{attribute 'GeneratedUsingTerminal: EK1100-0000-0018'}
{attribute addProperty BoxType "EK1100-0000-0018"}
{attribute addProperty Id "A_0014_BK1250_0000_0000A_0014_BK1250_0000_0000_09E1EB450"}
{attribute addProperty CRC "1503947044"}
{attribute addProperty Size "0"}
TYPE Beckhoff_BKxxxxsub_EK1100_59A46924 EXTENDS EK1100_1FC0878B :
STRUCT
	{attribute addProperty Name "A_0014_BK1250_0000_0000"}
	A_0014_BK1250_0000_0000 : A_0014_BK1250_0000_0000_09E1EB45;
END_STRUCT
END_TYPE

(* stored: Version 1.2.0.0, ProductVersion 3.1.4024.9
   DUT Beckhoff_BKxxxxsub_EK1100_59A46924: Id {f4793c22-162d-46d7-95b0-5ea1c2ce9a60} *)
